ADAPTER QueryServicesAdp (* Query services adapter *)
  (* Standard: 61499-2; Description: Copyright (c) 2018 fortiss GmbH This program and the accompanying materials are made available under the terms of the Eclipse Public License 2.0 which is available at https://www.eclipse.org/legal/epl-2.0/ SPDX-License-Identifier: EPL-2.0 *)
  (* Version 1.0, 2018-09-21, Jose Cabral, fortiss GmbH *)
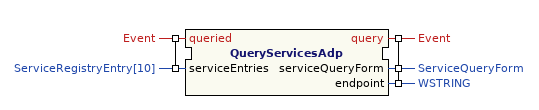
  EVENT_INPUT
    queried WITH serviceEntries; (* Query finished *)
  END_EVENT
  EVENT_OUTPUT
    query WITH serviceQueryForm, endpoint; (* Query for services *)
  END_EVENT
  VAR_INPUT
    serviceEntries : ARRAY [0..9] OF ServiceRegistryEntry; (* Result of the query request *)
  END_VAR
  VAR_OUTPUT
    serviceQueryForm : ServiceQueryForm; (* The Arrowhead Service object that is looked for (SD and supported IDD-s) *)
    endpoint : WSTRING; (* Endpoint (IP:PORT/URI) of the Service Registry (not officially in the documentation, but it simplifies the FBs) *)
  END_VAR
  (* Service SOCKET/PLUG: Query services adapter *)
END_ADAPTER
